// TIA Portal V17 export
// export: Created 2026-05-13T15:30:41.7173255Z, ExportSetting WithDefaults, DisplayName Totally Integrated Automation Portal, DisplayVersion V17 Update 4, DisplayName TIA Portal Openness, DisplayVersion V17 Update 4, DisplayName TIA Portal Version Control Interface, DisplayVersion V17, DisplayName SINAMICS Startdrive Advanced, DisplayVersion V17, DisplayName SINAMICS Startdrive G130, G150, S120, S150, SINAMICS MV, S210, DisplayVersion V17, DisplayName SINAMICS Startdrive G110M, G120, G120C, G120D, G120P, G115D, DisplayVersion V17, DisplayName STEP 7 Professional, DisplayVersion V17 Update 4, DisplayName STEP 7 Safety, DisplayVersion V17, DisplayName WinCC Professional, DisplayVersion V17 Update 4
TagTable "Codex_Popup_Sim_Int_Tags"
  Sim_SelectedCompID : Int  (1 s, start 1)   // Selected component ID. 1=Valve01, 2=Heater01, 3=Fan01.
  Sim_ClickPulse : Int  (1 s, start 0)   // Component click trigger pulse.
  Sim_DoubleClickTime_ms : Int  (1 s, start 800)   // Double-click time in milliseconds.
  Sim_Switch1 : Int  (1 s, start 0)   // Simulated Switch[1].
  Sim_RealValue1_Int : Int  (1 s, start 0)   // Integer placeholder for RealValue[1] simulation.
  Sim_Visible : Int  (1 s, start 0)   // Popup visible state.
  Sim_ActiveID : Int  (1 s, start 0)   // Current active popup ID.
  Sim_Confirmed : Int  (1 s, start 0)   // Confirmed state.
  Sim_ConfirmPulse : Int  (1 s, start 0)   // Confirm button pulse.
  Sim_CancelPulse : Int  (1 s, start 0)   // Cancel button pulse.
